FUNCTION_BLOCK FB_ModbusMaster //IMPLEMENTS I_UniversalUnit
VAR
	sName			:		STRING;
	bInitialized	:		BOOL;
	iScantime		:		UINT;
	iTimeout		:		UINT;
	//iErrorID		:		UDINT;
	iErrorID		:		MODBUS_ERRORS;
	
	bBusy			: 		BOOL;
	bError			:		BOOL;
	
	iStepInit		:		INT;
	iStepGeneral	: 		INT;
	iStepRunning	:		INT;
	bFirstCycle		:		BOOL;
	
	bRun			:		BOOL;
	bStop			: 		BOOL;
	
//	fbModbusMaster	: 		ModbusRtuMaster_PcCOM;
	fbModbusMaster : 		ModbusRtuMaster_KL6x22B;
	ipModbusSlave	:		ARRAY [1..247] OF I_ModbusSlave;
	iAmountSlave	: 		UINT;
	
	iLoopSlave		:		UINT	:= 1;
	iLoopAdr		:		UINT;
	iQuantity 		: 		POINTER TO WORD;
	iMBAddr 		: 		POINTER TO WORD;
    arrData			: 		ARRAY [0..255] OF BYTE;
	
	bDelayState		:		BOOL;
	tonScanTime		:		TON;
	
	tonTest			: TON;
	
END_VAR

IF bFirstCycle THEN
	bFirstCycle := FALSE;
END_IF
		
StateMachine();

bRun := FALSE;
bStop := FALSE;

bInitialized := iStepGeneral >= 20;
bBusy := fbModbusMaster.BUSY AND iStepGeneral = 30;

bError S= fbModbusMaster.Error AND iStepGeneral = 30 and iStepRunning = 60;
bError R= NOT fbModbusMaster.Error AND iStepGeneral = 30 AND iStepRunning = 60;
IF iStepGeneral = 30 AND iStepRunning = 60 THEN
	iErrorID := fbModbusMaster.ErrorId;
END_IF

tonScanTime(IN := iStepRunning >= 10 AND iStepRunning <= 60 AND iLoopSlave > iAmountSlave, PT := INT_TO_TIME(iScantime));

//	// error	
//		fbAxisError.Description := FUN_MergeStrings5(sMotorName, ' axis error number: ', UDINT_TO_STRING(iErrorID), '', '');
//		fbAxisError.Set(bError);

METHOD Abort : BOOL
END_METHOD

PROPERTY AnyError : BOOL
GET
AnyError 	:= bError;
END_GET
END_PROPERTY

PROPERTY Busy : BOOL
GET
Busy := bBusy;
END_GET
END_PROPERTY

PROPERTY ErrorID : UDINT
GET
ErrorID := iErrorID;
END_GET
END_PROPERTY

METHOD FirstCycle : BOOL
VAR_INPUT
//	ipAlarmController	: I_AlarmController;
//	ipHMIController	: I_HMIController;
END_VAR
END_METHOD

METHOD Init : BOOL
IF iStepGeneral = 0 THEN
	iStepGeneral := 10;
END_IF

//Method output
	Init := (iStepGeneral >= 20);
END_METHOD

PROPERTY Initialized : BOOL
GET
Initialized := bInitialized;
END_GET
END_PROPERTY

PROPERTY Name : STRING
GET
Name := sName;
END_GET
SET
sName := Name;
END_SET
END_PROPERTY

PROPERTY ReadData : ARRAY [0..255] OF BYTE
GET
ReadData := arrData;
END_GET
END_PROPERTY

PROPERTY ReadDataSize : uint
GET
ReadDataSize := INT_TO_UINT(SIZEOF(arrData));
END_GET
END_PROPERTY

METHOD RegisterSlave : BOOL
VAR_INPUT
	ModbusSlave		:		I_ModbusSlave;
END_VAR
VAR
	iLoop	:	UINT;
	bExists	:	BOOL;
END_VAR
FOR iLoop := 1 TO iAmountSlave DO
	IF ipModbusSlave[iLoop] = ModbusSlave THEN
		bExists := TRUE;
		iLoop := iAmountSlave;
	END_IF
END_FOR 
IF NOT bExists THEN
	iAmountSlave := iAmountSlave + 1;
	ipModbusSlave[iAmountSlave] := ModbusSlave;
END_IF
END_METHOD

METHOD Reset : BOOL
bError := FALSE;
iErrorID := 0;
bError := FALSE;
iStepInit		:= 0;
iStepGeneral	:= 0;
iStepRunning	:= 0;

iLoopSlave		:= 1;
iLoopAdr		:= 0;

fbModbusMaster.Execute := FALSE;

Reset := TRUE;
END_METHOD

METHOD Run : BOOL
IF (iStepGeneral = 20) THEN
	iStepGeneral := 30;
END_IF

bRun := TRUE;
Run := (iStepGeneral >= 30) AND (iStepGeneral < 200);
END_METHOD

PROPERTY ScanTime : UINT
GET
ScanTime := iScantime;
END_GET
SET
iScantime := ScanTime;
END_SET
END_PROPERTY

METHOD StateInit : BOOL (*Unit is performing initialization*)
IF NOT bError THEN
	iStepGeneral := 20;
END_IF
END_METHOD

METHOD StateMachine : BOOL (*State machine of unit*)
//State machine						   
	CASE iStepGeneral OF
		0:  //Uninitialized
			StateUninitialized();
	
		10: //Initializing
			StateInit();
	
		20: //Ready
			StateReady();
		
		30: //Running
			StateRunning();
						
		200: //stop
			StateStopping();
			
		210: //stop done
			StateStoppingDone();
	END_CASE
END_METHOD

METHOD StateReady : BOOL (* Unit is initialized*)
END_METHOD

METHOD StateRunning : BOOL (* Unit is uninitialized*)
VAR 
END_VAR
CASE iStepRunning OF
	0: // Trigger
		IF iAmountSlave > 0 THEN
			iStepRunning := 10;
		ELSE
			iStepRunning := 50;
		END_IF
		
	10: // Set parameters
		IF iLoopSlave <= iAmountSlave THEN
			IF  iLoopAdr <= ipModbusSlave[iLoopSlave].NumAddRegion - 1 THEN
				iQuantity := (ipModbusSlave[iLoopSlave].Address + (iLoopAdr*2+1)*SIZEOF(WORD));
				iMBAddr := (ipModbusSlave[iLoopSlave].Address + (iLoopAdr*2)*SIZEOF(WORD));
				
				fbModbusMaster.UnitID 	:=		ipModbusSlave[iLoopSlave].UnitID;
				fbModbusMaster.Quantity	:=		iQuantity^;
				fbModbusMaster.MBAddr	:=		iMBAddr^;
				fbModbusMaster.cbLength	:= 		SIZEOF(arrData);
				fbModbusMaster.pMemoryAddr	:= 	ADR(arrData);
				fbModbusMaster.Timeout	:= 		UINT_TO_TIME(iTimeout);
				
				iLoopAdr := iLoopAdr + 1;
				iStepRunning := 20;
			ELSE
				iLoopAdr := 0;
				iLoopSlave := iLoopSlave + 1;
				iStepRunning := 60;
				bDelayState := NOT bDelayState;
			END_IF
		ELSE
			iLoopSlave := 1;
			iStepRunning := 60;
			bDelayState := NOT bDelayState;
		END_IF
		
	20: // Send request
		IF NOT fbModbusMaster.BUSY THEN
			iStepRunning := 30;
		END_IF
	
	30: // Wait ack request
		IF fbModbusMaster.BUSY THEN
			iStepRunning := 40;
		END_IF
		
	40: // Wait respond
		IF NOT fbModbusMaster.BUSY THEN
			iStepRunning := 50;
		END_IF
		
	50: // Convert raw data
		IF iLoopSlave <= iAmountSlave THEN
			ipModbusSlave[iLoopSlave].Convert(iLoopAdr, ADR(arrData));
		END_IF
		bDelayState := NOT bDelayState;
//		IF tonTest.Q  THEN
			iStepRunning := 60;
//		END_IF


	60: // Return, done
		IF NOT bDelayState AND tonScanTime.Q THEN
			iStepRunning := 0;
		END_IF
		bDelayState := NOT bDelayState;
		
END_CASE

IF (iStepRunning >= 20) AND (iStepRunning <= 40) THEN
	fbModbusMaster.ReadRegs();
END_IF
fbModbusMaster.Execute := iStepRunning >= 20 AND iStepRunning <= 30;
tonTest(IN := iStepRunning = 50, PT := T#2S);
END_METHOD

METHOD StateStopping : BOOL (* Unit is uninitialized*)
iStepGeneral	:= 210;
iStepRunning	:= 0;

iLoopSlave		:= 1;
iLoopAdr		:= 0;

fbModbusMaster.Execute := FALSE;
END_METHOD

METHOD StateStoppingDone : BOOL (* Unit is uninitialized*)
IF NOT bStop THEN
	iStepGeneral := 20;
END_IF
END_METHOD

METHOD StateUninitialized : BOOL (* Unit is uninitialized*)
END_METHOD

METHOD Stop : BOOL
IF iStepGeneral >= 30 AND iStepGeneral < 200 THEN
	iStepGeneral := 200;
END_IF
bStop := TRUE;

Stop := (iStepGeneral = 210);
END_METHOD

PROPERTY Timeout : UINT
GET
Timeout := iTimeout;
END_GET
SET
iTimeout := Timeout;
END_SET
END_PROPERTY

END_FUNCTION_BLOCK

(* stored: Version 1.1.0.1, ProductVersion 3.1.4024.12
   POU FB_ModbusMaster: Id {383531aa-3652-4615-9883-854b84ebdc31}, SpecialFunc None
   Folder Methods: Id {067e956d-7447-440b-bb7c-a17eb17d60b1}
   Folder Properties: Id {dda8d42f-2796-433c-8b44-7c0e273aa52f}
   Folder StateMachine: Id {58b557b7-d2c2-457b-a8d0-dbac8b324ebc}
   Method Abort: Id {d170ce10-c663-4dfe-9dba-a085107ba388}
   Property AnyError: Id {45cb1e5b-801a-4c7d-a80e-9506285dfb3c}
   Get Get: Id {360cff8f-569b-4317-8045-69ce24908b7f}
   Property Busy: Id {b11648ea-ec4e-40e9-adc4-f77827ee7f01}
   Get Get: Id {a1c5374b-3865-4838-b65b-f5c6a0835665}
   Property ErrorID: Id {81dab0ad-62e0-4fd2-94f4-3786bdfc5c61}
   Get Get: Id {bd49841c-7579-429c-bb3e-55f6c8382d66}
   Method FirstCycle: Id {b81bd56c-9f95-4518-88ea-14ab1af8620f}
   Method Init: Id {adb0f840-9854-48bb-9867-8558f3fc8764}
   Property Initialized: Id {2f2b00e9-f2c5-40fe-be3e-593bf36d21e2}
   Get Get: Id {7101007d-b47d-47a8-8511-547d82564dfb}
   Property Name: Id {f8832320-307e-488d-ba14-68e6271ef348}
   Get Get: Id {10c882c2-26e5-4d65-9bcc-3499aabfe3c5}
   Set Set: Id {015f49a9-8a42-4718-b2c7-58ce03a742aa}
   Property ReadData: Id {75712a42-a84c-4947-ac2a-2d1b25b7b297}
   Get Get: Id {95024ca2-66ad-4b16-920e-6d1ddd469ac1}
   Property ReadDataSize: Id {3cb8fabd-08bb-4c22-96b3-af7830849c39}
   Get Get: Id {a8dc376e-955f-46b6-9b33-957335fbc210}
   Method RegisterSlave: Id {991fe131-bc6d-4e7e-9414-d4034de09ad3}
   Method Reset: Id {4190b5ad-ee32-41e6-86da-3cf60dfcd435}
   Method Run: Id {07a8bc59-999b-4d59-9560-feef9f903a20}
   Property ScanTime: Id {5b7878c4-4362-4d5b-99fa-9da47a4ca446}
   Get Get: Id {541e4923-ad17-4562-a852-1c8367bee7da}
   Set Set: Id {87feb87e-b4e3-41e6-89af-09cc8001252c}
   Method StateInit: Id {4e49a1af-97ef-4ae6-a0c3-b5234cc2497a}
   Method StateMachine: Id {c5907cd4-9636-4b7b-9f9b-3b47835d586e}
   Method StateReady: Id {652bc040-6918-41f6-8573-0396ad5da8fa}
   Method StateRunning: Id {97a85ca0-cdf0-4a98-99b6-286d42d839ec}
   Method StateStopping: Id {a5bc9935-91a4-4fec-8e4d-82d2573de05f}
   Method StateStoppingDone: Id {d6ba127c-7dd9-4267-bb45-f2c5c72fb129}
   Method StateUninitialized: Id {02a14e5c-79b0-481c-be40-ba9ce91213fc}
   Method Stop: Id {d08751b9-9c58-450d-8b27-62019e485f78}
   Property Timeout: Id {ad915020-ee1a-4de9-9ab5-c123d6eefbc6}
   Get Get: Id {33cc4f60-c2e8-4a21-b4ee-4e39dcc2be36}
   Set Set: Id {b1706c38-23dd-439c-ad15-24cf2b70e594} *)
